// Dispositivo/Application/Pages/Schedulle
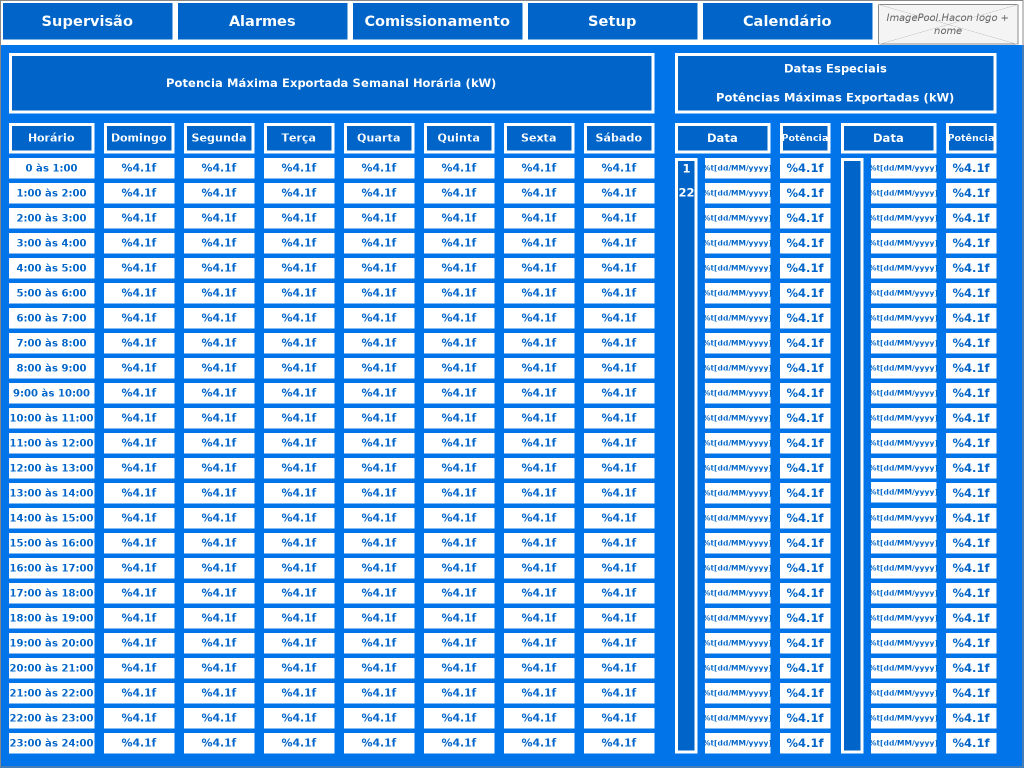
VISUALIZATION Schedulle  // 1024x768
    Frame (0,0 1024x768)
        shows Template()
    Rectangle (675,53 321x60), "Datas Especiais Potências Máximas Exportadas (kW)"
        OnMouseClick:  Assign=Setup, Type=Assignment
    Rectangle (104,123 70x30), "Domingo"
        OnMouseClick:  Assign=Setup, Type=Assignment
    Rectangle (104,158 70x20), "%4.1f", text variable: PerVar.WeekSchedule_kW[1,1]
        OnMouseEnter: write the text variable via Default, min 0, max 5000
    Rectangle (104,183 70x20), "%4.1f", text variable: PerVar.WeekSchedule_kW[1,2]
        OnMouseEnter: write the text variable via Default, min 0, max 5000
    Rectangle (104,208 70x20), "%4.1f", text variable: PerVar.WeekSchedule_kW[1,3]
        OnMouseEnter: write the text variable via Default, min 0, max 5000
    Rectangle (104,233 70x20), "%4.1f", text variable: PerVar.WeekSchedule_kW[1,4]
        OnMouseEnter: write the text variable via Default, min 0, max 5000
    Rectangle (104,258 70x20), "%4.1f", text variable: PerVar.WeekSchedule_kW[1,5]
        OnMouseEnter: write the text variable via Default, min 0, max 5000
    Rectangle (104,283 70x20), "%4.1f", text variable: PerVar.WeekSchedule_kW[1,6]
        OnMouseEnter: write the text variable via Default, min 0, max 5000
    Rectangle (104,308 70x20), "%4.1f", text variable: PerVar.WeekSchedule_kW[1,7]
        OnMouseEnter: write the text variable via Default, min 0, max 5000
    Rectangle (104,333 70x20), "%4.1f", text variable: PerVar.WeekSchedule_kW[1,8]
        OnMouseEnter: write the text variable via Default, min 0, max 5000
    Rectangle (104,358 70x20), "%4.1f", text variable: PerVar.WeekSchedule_kW[1,9]
        OnMouseEnter: write the text variable via Default, min 0, max 5000
    Rectangle (104,383 70x20), "%4.1f", text variable: PerVar.WeekSchedule_kW[1,10]
        OnMouseEnter: write the text variable via Default, min 0, max 5000
    Rectangle (104,408 70x20), "%4.1f", text variable: PerVar.WeekSchedule_kW[1,11]
        OnMouseEnter: write the text variable via Default, min 0, max 5000
    Rectangle (104,433 70x20), "%4.1f", text variable: PerVar.WeekSchedule_kW[1,12]
        OnMouseEnter: write the text variable via Default, min 0, max 5000
    Rectangle (104,458 70x20), "%4.1f", text variable: PerVar.WeekSchedule_kW[1,13]
        OnMouseEnter: write the text variable via Default, min 0, max 5000
    Rectangle (104,483 70x20), "%4.1f", text variable: PerVar.WeekSchedule_kW[1,14]
        OnMouseEnter: write the text variable via Default, min 0, max 5000
    Rectangle (104,508 70x20), "%4.1f", text variable: PerVar.WeekSchedule_kW[1,15]
        OnMouseEnter: write the text variable via Default, min 0, max 5000
    Rectangle (104,533 70x20), "%4.1f", text variable: PerVar.WeekSchedule_kW[1,16]
        OnMouseEnter: write the text variable via Default, min 0, max 5000
    Rectangle (104,558 70x20), "%4.1f", text variable: PerVar.WeekSchedule_kW[1,17]
        OnMouseEnter: write the text variable via Default, min 0, max 5000
    Rectangle (104,583 70x20), "%4.1f", text variable: PerVar.WeekSchedule_kW[1,18]
        OnMouseEnter: write the text variable via Default, min 0, max 5000
    Rectangle (104,608 70x20), "%4.1f", text variable: PerVar.WeekSchedule_kW[1,19]
        OnMouseEnter: write the text variable via Default, min 0, max 5000
    Rectangle (104,633 70x20), "%4.1f", text variable: PerVar.WeekSchedule_kW[1,20]
        OnMouseEnter: write the text variable via Default, min 0, max 5000
    Rectangle (104,658 70x20), "%4.1f", text variable: PerVar.WeekSchedule_kW[1,21]
        OnMouseEnter: write the text variable via Default, min 0, max 5000
    Rectangle (104,683 70x20), "%4.1f", text variable: PerVar.WeekSchedule_kW[1,22]
        OnMouseEnter: write the text variable via Default, min 0, max 5000
    Rectangle (104,708 70x20), "%4.1f", text variable: PerVar.WeekSchedule_kW[1,23]
        OnMouseEnter: write the text variable via Default, min 0, max 5000
    Rectangle (104,733 70x20), "%4.1f", text variable: PerVar.WeekSchedule_kW[1,24]
        OnMouseEnter: write the text variable via Default, min 0, max 5000
    Rectangle (705,158 65x20), "%t[dd/MM/yyyy]", tooltip "XX/XX/XXXX", text variable: PerVar.DatasEspeciais[1]
        OnMouseClick: write the text variable via Edit
    Rectangle (675,123 95x30), "Data"
        OnMouseClick:  Assign=Setup, Type=Assignment
    Rectangle (705,183 65x20), "%t[dd/MM/yyyy]", tooltip "XX/XX/XXXX", text variable: PerVar.DatasEspeciais[2]
        OnMouseClick: write the text variable via Edit
    Rectangle (705,208 65x20), "%t[dd/MM/yyyy]", tooltip "XX/XX/XXXX", text variable: PerVar.DatasEspeciais[3]
        OnMouseClick: write the text variable via Edit
    Rectangle (705,233 65x20), "%t[dd/MM/yyyy]", tooltip "XX/XX/XXXX", text variable: PerVar.DatasEspeciais[4]
        OnMouseClick: write the text variable via Edit
    Rectangle (705,258 65x20), "%t[dd/MM/yyyy]", tooltip "XX/XX/XXXX", text variable: PerVar.DatasEspeciais[5]
        OnMouseClick: write the text variable via Edit
    Rectangle (705,283 65x20), "%t[dd/MM/yyyy]", tooltip "XX/XX/XXXX", text variable: PerVar.DatasEspeciais[6]
        OnMouseClick: write the text variable via Edit
    Rectangle (705,308 65x20), "%t[dd/MM/yyyy]", tooltip "XX/XX/XXXX", text variable: PerVar.DatasEspeciais[7]
        OnMouseClick: write the text variable via Edit
    Rectangle (705,333 65x20), "%t[dd/MM/yyyy]", tooltip "XX/XX/XXXX", text variable: PerVar.DatasEspeciais[8]
        OnMouseClick: write the text variable via Edit
    Rectangle (705,358 65x20), "%t[dd/MM/yyyy]", tooltip "XX/XX/XXXX", text variable: PerVar.DatasEspeciais[9]
        OnMouseClick: write the text variable via Edit
    Rectangle (705,383 65x20), "%t[dd/MM/yyyy]", tooltip "XX/XX/XXXX", text variable: PerVar.DatasEspeciais[10]
        OnMouseClick: write the text variable via Edit
    Rectangle (705,408 65x20), "%t[dd/MM/yyyy]", tooltip "XX/XX/XXXX", text variable: PerVar.DatasEspeciais[11]
        OnMouseClick: write the text variable via Edit
    Rectangle (705,433 65x20), "%t[dd/MM/yyyy]", tooltip "XX/XX/XXXX", text variable: PerVar.DatasEspeciais[12]
        OnMouseClick: write the text variable via Edit
    Rectangle (705,458 65x20), "%t[dd/MM/yyyy]", tooltip "XX/XX/XXXX", text variable: PerVar.DatasEspeciais[13]
        OnMouseClick: write the text variable via Edit
    Rectangle (705,483 65x20), "%t[dd/MM/yyyy]", tooltip "XX/XX/XXXX", text variable: PerVar.DatasEspeciais[14]
        OnMouseClick: write the text variable via Edit
    Rectangle (705,508 65x20), "%t[dd/MM/yyyy]", tooltip "XX/XX/XXXX", text variable: PerVar.DatasEspeciais[15]
        OnMouseClick: write the text variable via Edit
    Rectangle (841,123 95x30), "Data"
        OnMouseClick:  Assign=Setup, Type=Assignment
    Rectangle (871,158 65x20), "%t[dd/MM/yyyy]", tooltip "XX/XX/XXXX", text variable: PerVar.DatasEspeciais[25]
        OnMouseClick: write the text variable via Edit
    Rectangle (871,183 65x20), "%t[dd/MM/yyyy]", tooltip "XX/XX/XXXX", text variable: PerVar.DatasEspeciais[26]
        OnMouseClick: write the text variable via Edit
    Rectangle (871,208 65x20), "%t[dd/MM/yyyy]", tooltip "XX/XX/XXXX", text variable: PerVar.DatasEspeciais[27]
        OnMouseClick: write the text variable via Edit
    Rectangle (871,233 65x20), "%t[dd/MM/yyyy]", tooltip "XX/XX/XXXX", text variable: PerVar.DatasEspeciais[28]
        OnMouseClick: write the text variable via Edit
    Rectangle (871,258 65x20), "%t[dd/MM/yyyy]", tooltip "XX/XX/XXXX", text variable: PerVar.DatasEspeciais[29]
        OnMouseClick: write the text variable via Edit
    Rectangle (871,283 65x20), "%t[dd/MM/yyyy]", tooltip "XX/XX/XXXX", text variable: PerVar.DatasEspeciais[30]
        OnMouseClick: write the text variable via Edit
    Rectangle (871,308 65x20), "%t[dd/MM/yyyy]", tooltip "XX/XX/XXXX", text variable: PerVar.DatasEspeciais[31]
        OnMouseClick: write the text variable via Edit
    Rectangle (871,333 65x20), "%t[dd/MM/yyyy]", tooltip "XX/XX/XXXX", text variable: PerVar.DatasEspeciais[32]
        OnMouseClick: write the text variable via Edit
    Rectangle (871,358 65x20), "%t[dd/MM/yyyy]", tooltip "XX/XX/XXXX", text variable: PerVar.DatasEspeciais[33]
        OnMouseClick: write the text variable via Edit
    Rectangle (871,383 65x20), "%t[dd/MM/yyyy]", tooltip "XX/XX/XXXX", text variable: PerVar.DatasEspeciais[34]
        OnMouseClick: write the text variable via Edit
    Rectangle (871,408 65x20), "%t[dd/MM/yyyy]", tooltip "XX/XX/XXXX", text variable: PerVar.DatasEspeciais[35]
        OnMouseClick: write the text variable via Edit
    Rectangle (871,433 65x20), "%t[dd/MM/yyyy]", tooltip "XX/XX/XXXX", text variable: PerVar.DatasEspeciais[36]
        OnMouseClick: write the text variable via Edit
    Rectangle (871,458 65x20), "%t[dd/MM/yyyy]", tooltip "XX/XX/XXXX", text variable: PerVar.DatasEspeciais[37]
        OnMouseClick: write the text variable via Edit
    Rectangle (871,482 65x20), "%t[dd/MM/yyyy]", tooltip "XX/XX/XXXX", text variable: PerVar.DatasEspeciais[38]
        OnMouseClick: write the text variable via Edit
    Rectangle (871,508 65x20), "%t[dd/MM/yyyy]", tooltip "XX/XX/XXXX", text variable: PerVar.DatasEspeciais[39]
        OnMouseClick: write the text variable via Edit
    Rectangle (780,123 50x30), "Potência"
        OnMouseClick:  Assign=Setup, Type=Assignment
    Rectangle (780,158 50x20), "%4.1f", text variable: PerVar.SpecialDaySchedule[1]
        OnMouseEnter: write the text variable via Default, min 0, max 5000
    Rectangle (780,183 50x20), "%4.1f", text variable: PerVar.SpecialDaySchedule[2]
        OnMouseEnter: write the text variable via Default, min 0, max 5000
    Rectangle (780,208 50x20), "%4.1f", text variable: PerVar.SpecialDaySchedule[3]
        OnMouseEnter: write the text variable via Default, min 0, max 5000
    Rectangle (780,233 50x20), "%4.1f", text variable: PerVar.SpecialDaySchedule[4]
        OnMouseEnter: write the text variable via Default, min 0, max 5000
    Rectangle (780,258 50x20), "%4.1f", text variable: PerVar.SpecialDaySchedule[5]
        OnMouseEnter: write the text variable via Default, min 0, max 5000
    Rectangle (780,283 50x20), "%4.1f", text variable: PerVar.SpecialDaySchedule[6]
        OnMouseEnter: write the text variable via Default, min 0, max 5000
    Rectangle (780,308 50x20), "%4.1f", text variable: PerVar.SpecialDaySchedule[7]
        OnMouseEnter: write the text variable via Default, min 0, max 5000
    Rectangle (780,333 50x20), "%4.1f", text variable: PerVar.SpecialDaySchedule[8]
        OnMouseEnter: write the text variable via Default, min 0, max 5000
    Rectangle (780,358 50x20), "%4.1f", text variable: PerVar.SpecialDaySchedule[9]
        OnMouseEnter: write the text variable via Default, min 0, max 5000
    Rectangle (780,383 50x20), "%4.1f", text variable: PerVar.SpecialDaySchedule[10]
        OnMouseEnter: write the text variable via Default, min 0, max 5000
    Rectangle (780,408 50x20), "%4.1f", text variable: PerVar.SpecialDaySchedule[11]
        OnMouseEnter: write the text variable via Default, min 0, max 5000
    Rectangle (780,433 50x20), "%4.1f", text variable: PerVar.SpecialDaySchedule[12]
        OnMouseEnter: write the text variable via Default, min 0, max 5000
    Rectangle (780,458 50x20), "%4.1f", text variable: PerVar.SpecialDaySchedule[13]
        OnMouseEnter: write the text variable via Default, min 0, max 5000
    Rectangle (780,483 50x20), "%4.1f", text variable: PerVar.SpecialDaySchedule[14]
        OnMouseEnter: write the text variable via Default, min 0, max 5000
    Rectangle (780,508 50x20), "%4.1f", text variable: PerVar.SpecialDaySchedule[15]
        OnMouseEnter: write the text variable via Default, min 0, max 5000
    Rectangle (780,533 50x20), "%4.1f", text variable: PerVar.SpecialDaySchedule[16]
        OnMouseEnter: write the text variable via Default, min 0, max 5000
    Rectangle (780,558 50x20), "%4.1f", text variable: PerVar.SpecialDaySchedule[17]
        OnMouseEnter: write the text variable via Default, min 0, max 5000
    Rectangle (780,583 50x20), "%4.1f", text variable: PerVar.SpecialDaySchedule[18]
        OnMouseEnter: write the text variable via Default, min 0, max 5000
    Rectangle (780,608 50x20), "%4.1f", text variable: PerVar.SpecialDaySchedule[19]
        OnMouseEnter: write the text variable via Default, min 0, max 5000
    Rectangle (780,633 50x20), "%4.1f", text variable: PerVar.SpecialDaySchedule[20]
        OnMouseEnter: write the text variable via Default, min 0, max 5000
    Rectangle (780,658 50x20), "%4.1f", text variable: PerVar.SpecialDaySchedule[21]
        OnMouseEnter: write the text variable via Default, min 0, max 5000
    Rectangle (780,683 50x20), "%4.1f", text variable: PerVar.SpecialDaySchedule[22]
        OnMouseEnter: write the text variable via Default, min 0, max 5000
    Rectangle (780,708 50x20), "%4.1f", text variable: PerVar.SpecialDaySchedule[23]
        OnMouseEnter: write the text variable via Default, min 0, max 5000
    Rectangle (780,733 50x20), "%4.1f", text variable: PerVar.SpecialDaySchedule[24]
        OnMouseEnter: write the text variable via Default, min 0, max 5000
    Rectangle (946,158 50x20), "%4.1f", text variable: PerVar.SpecialDaySchedule[25]
        OnMouseEnter: write the text variable via Default, min 0, max 5000
    Rectangle (946,183 50x20), "%4.1f", text variable: PerVar.SpecialDaySchedule[26]
        OnMouseEnter: write the text variable via Default, min 0, max 5000
    Rectangle (946,208 50x20), "%4.1f", text variable: PerVar.SpecialDaySchedule[27]
        OnMouseEnter: write the text variable via Default, min 0, max 5000
    Rectangle (946,233 50x20), "%4.1f", text variable: PerVar.SpecialDaySchedule[28]
        OnMouseEnter: write the text variable via Default, min 0, max 5000
    Rectangle (946,258 50x20), "%4.1f", text variable: PerVar.SpecialDaySchedule[29]
        OnMouseEnter: write the text variable via Default, min 0, max 5000
    Rectangle (946,283 50x20), "%4.1f", text variable: PerVar.SpecialDaySchedule[30]
        OnMouseEnter: write the text variable via Default, min 0, max 5000
    Rectangle (705,533 65x20), "%t[dd/MM/yyyy]", tooltip "XX/XX/XXXX", text variable: PerVar.DatasEspeciais[16]
        OnMouseClick: write the text variable via Edit
    Rectangle (705,558 65x20), "%t[dd/MM/yyyy]", tooltip "XX/XX/XXXX", text variable: PerVar.DatasEspeciais[17]
        OnMouseClick: write the text variable via Edit
    Rectangle (705,583 65x20), "%t[dd/MM/yyyy]", tooltip "XX/XX/XXXX", text variable: PerVar.DatasEspeciais[18]
        OnMouseClick: write the text variable via Edit
    Rectangle (705,608 65x20), "%t[dd/MM/yyyy]", tooltip "XX/XX/XXXX", text variable: PerVar.DatasEspeciais[19]
        OnMouseClick: write the text variable via Edit
    Rectangle (705,633 65x20), "%t[dd/MM/yyyy]", tooltip "XX/XX/XXXX", text variable: PerVar.DatasEspeciais[20]
        OnMouseClick: write the text variable via Edit
    Rectangle (705,658 65x20), "%t[dd/MM/yyyy]", tooltip "XX/XX/XXXX", text variable: PerVar.DatasEspeciais[21]
        OnMouseClick: write the text variable via Edit
    Rectangle (705,683 65x20), "%t[dd/MM/yyyy]", tooltip "XX/XX/XXXX", text variable: PerVar.DatasEspeciais[22]
        OnMouseClick: write the text variable via Edit
    Rectangle (705,708 65x20), "%t[dd/MM/yyyy]", tooltip "XX/XX/XXXX", text variable: PerVar.DatasEspeciais[23]
        OnMouseClick: write the text variable via Edit
    Rectangle (705,733 65x20), "%t[dd/MM/yyyy]", tooltip "XX/XX/XXXX", text variable: PerVar.DatasEspeciais[24]
        OnMouseClick: write the text variable via Edit
    Rectangle (871,533 65x20), "%t[dd/MM/yyyy]", tooltip "XX/XX/XXXX", text variable: PerVar.DatasEspeciais[40]
        OnMouseClick: write the text variable via Edit
    Rectangle (871,558 65x20), "%t[dd/MM/yyyy]", tooltip "XX/XX/XXXX", text variable: PerVar.DatasEspeciais[41]
        OnMouseClick: write the text variable via Edit
    Rectangle (871,583 65x20), "%t[dd/MM/yyyy]", tooltip "XX/XX/XXXX", text variable: PerVar.DatasEspeciais[42]
        OnMouseClick: write the text variable via Edit
    Rectangle (871,608 65x20), "%t[dd/MM/yyyy]", tooltip "XX/XX/XXXX", text variable: PerVar.DatasEspeciais[43]
        OnMouseClick: write the text variable via Edit
    Rectangle (871,633 65x20), "%t[dd/MM/yyyy]", tooltip "XX/XX/XXXX", text variable: PerVar.DatasEspeciais[44]
        OnMouseClick: write the text variable via Edit
    Rectangle (871,658 65x20), "%t[dd/MM/yyyy]", tooltip "XX/XX/XXXX", text variable: PerVar.DatasEspeciais[45]
        OnMouseClick: write the text variable via Edit
    Rectangle (871,683 65x20), "%t[dd/MM/yyyy]", tooltip "XX/XX/XXXX", text variable: PerVar.DatasEspeciais[46]
        OnMouseClick: write the text variable via Edit
    Rectangle (871,708 65x20), "%t[dd/MM/yyyy]", tooltip "XX/XX/XXXX", text variable: PerVar.DatasEspeciais[47]
        OnMouseClick: write the text variable via Edit
    Rectangle (871,733 65x20), "%t[dd/MM/yyyy]", tooltip "XX/XX/XXXX", text variable: PerVar.DatasEspeciais[48]
        OnMouseClick: write the text variable via Edit
    Rectangle (946,308 50x20), "%4.1f", text variable: PerVar.SpecialDaySchedule[31]
        OnMouseEnter: write the text variable via Default, min 0, max 5000
    Rectangle (946,333 50x20), "%4.1f", text variable: PerVar.SpecialDaySchedule[32]
        OnMouseEnter: write the text variable via Default, min 0, max 5000
    Rectangle (946,358 50x20), "%4.1f", text variable: PerVar.SpecialDaySchedule[33]
        OnMouseEnter: write the text variable via Default, min 0, max 5000
    Rectangle (946,383 50x20), "%4.1f", text variable: PerVar.SpecialDaySchedule[34]
        OnMouseEnter: write the text variable via Default, min 0, max 5000
    Rectangle (946,408 50x20), "%4.1f", text variable: PerVar.SpecialDaySchedule[35]
        OnMouseEnter: write the text variable via Default, min 0, max 5000
    Rectangle (946,433 50x20), "%4.1f", text variable: PerVar.SpecialDaySchedule[36]
        OnMouseEnter: write the text variable via Default, min 0, max 5000
    Rectangle (946,458 50x20), "%4.1f", text variable: PerVar.SpecialDaySchedule[37]
        OnMouseEnter: write the text variable via Default, min 0, max 5000
    Rectangle (946,483 50x20), "%4.1f", text variable: PerVar.SpecialDaySchedule[38]
        OnMouseEnter: write the text variable via Default, min 0, max 5000
    Rectangle (946,508 50x20), "%4.1f", text variable: PerVar.SpecialDaySchedule[39]
        OnMouseEnter: write the text variable via Default, min 0, max 5000
    Rectangle (946,533 50x20), "%4.1f", text variable: PerVar.SpecialDaySchedule[40]
        OnMouseEnter: write the text variable via Default, min 0, max 5000
    Rectangle (946,558 50x20), "%4.1f", text variable: PerVar.SpecialDaySchedule[41]
        OnMouseEnter: write the text variable via Default, min 0, max 5000
    Rectangle (946,583 50x20), "%4.1f", text variable: PerVar.SpecialDaySchedule[42]
        OnMouseEnter: write the text variable via Default, min 0, max 5000
    Rectangle (946,608 50x20), "%4.1f", text variable: PerVar.SpecialDaySchedule[43]
        OnMouseEnter: write the text variable via Default, min 0, max 5000
    Rectangle (946,633 50x20), "%4.1f", text variable: PerVar.SpecialDaySchedule[44]
        OnMouseEnter: write the text variable via Default, min 0, max 5000
    Rectangle (946,658 50x20), "%4.1f", text variable: PerVar.SpecialDaySchedule[45]
        OnMouseEnter: write the text variable via Default, min 0, max 5000
    Rectangle (946,683 50x20), "%4.1f", text variable: PerVar.SpecialDaySchedule[46]
        OnMouseEnter: write the text variable via Default, min 0, max 5000
    Rectangle (946,708 50x20), "%4.1f", text variable: PerVar.SpecialDaySchedule[47]
        OnMouseEnter: write the text variable via Default, min 0, max 5000
    Rectangle (946,733 50x20), "%4.1f", text variable: PerVar.SpecialDaySchedule[48]
        OnMouseEnter: write the text variable via Default, min 0, max 5000
    Rectangle (9,53 645x60), "Potencia Máxima Exportada Semanal Horária (kW)"
        OnMouseClick:  Assign=Setup, Type=Assignment
    Rectangle (184,123 70x30), "Segunda"
        OnMouseClick:  Assign=Setup, Type=Assignment
    Rectangle (264,123 70x30), "Terça"
        OnMouseClick:  Assign=Setup, Type=Assignment
    Rectangle (344,123 70x30), "Quarta"
        OnMouseClick:  Assign=Setup, Type=Assignment
    Rectangle (424,123 70x30), "Quinta"
        OnMouseClick:  Assign=Setup, Type=Assignment
    Rectangle (504,123 70x30), "Sexta"
        OnMouseClick:  Assign=Setup, Type=Assignment
    Rectangle (584,123 70x30), "Sábado"
        OnMouseClick:  Assign=Setup, Type=Assignment
    Rectangle (9,158 85x20), "0 às 1:00"
    Rectangle (9,123 85x30), "Horário"
        OnMouseClick:  Assign=Setup, Type=Assignment
    Rectangle (9,183 85x20), "1:00 às 2:00"
    Rectangle (9,208 85x20), "2:00 às 3:00"
    Rectangle (9,233 85x20), "3:00 às 4:00"
    Rectangle (9,258 85x20), "4:00 às 5:00"
    Rectangle (9,283 85x20), "5:00 às 6:00"
    Rectangle (9,308 85x20), "6:00 às 7:00"
    Rectangle (9,333 85x20), "7:00 às 8:00"
    Rectangle (9,358 85x20), "8:00 às 9:00"
    Rectangle (9,383 85x20), "9:00 às 10:00"
    Rectangle (9,408 85x20), "10:00 às 11:00"
    Rectangle (9,433 85x20), "11:00 às 12:00"
    Rectangle (9,458 85x20), "12:00 às 13:00"
    Rectangle (9,483 85x20), "13:00 às 14:00"
    Rectangle (9,508 85x20), "14:00 às 15:00"
    Rectangle (9,533 85x20), "15:00 às 16:00"
    Rectangle (9,558 85x20), "16:00 às 17:00"
    Rectangle (9,583 85x20), "17:00 às 18:00"
    Rectangle (9,608 85x20), "18:00 às 19:00"
    Rectangle (9,633 85x20), "19:00 às 20:00"
    Rectangle (9,658 85x20), "20:00 às 21:00"
    Rectangle (9,683 85x20), "21:00 às 22:00"
    Rectangle (9,708 85x20), "22:00 às 23:00"
    Rectangle (9,733 85x20), "23:00 às 24:00"
    Rectangle (184,158 70x20), "%4.1f", text variable: PerVar.WeekSchedule_kW[2,1]
        OnMouseEnter: write the text variable via Default, min 0, max 5000
    Rectangle (184,183 70x20), "%4.1f", text variable: PerVar.WeekSchedule_kW[2,2]
        OnMouseEnter: write the text variable via Default, min 0, max 5000
    Rectangle (184,208 70x20), "%4.1f", text variable: PerVar.WeekSchedule_kW[2,3]
        OnMouseEnter: write the text variable via Default, min 0, max 5000
    Rectangle (184,233 70x20), "%4.1f", text variable: PerVar.WeekSchedule_kW[2,4]
        OnMouseEnter: write the text variable via Default, min 0, max 5000
    Rectangle (184,258 70x20), "%4.1f", text variable: PerVar.WeekSchedule_kW[2,5]
        OnMouseEnter: write the text variable via Default, min 0, max 5000
    Rectangle (184,283 70x20), "%4.1f", text variable: PerVar.WeekSchedule_kW[2,6]
        OnMouseEnter: write the text variable via Default, min 0, max 5000
    Rectangle (184,308 70x20), "%4.1f", text variable: PerVar.WeekSchedule_kW[2,7]
        OnMouseEnter: write the text variable via Default, min 0, max 5000
    Rectangle (184,333 70x20), "%4.1f", text variable: PerVar.WeekSchedule_kW[2,8]
        OnMouseEnter: write the text variable via Default, min 0, max 5000
    Rectangle (184,358 70x20), "%4.1f", text variable: PerVar.WeekSchedule_kW[2,9]
        OnMouseEnter: write the text variable via Default, min 0, max 5000
    Rectangle (184,383 70x20), "%4.1f", text variable: PerVar.WeekSchedule_kW[2,10]
        OnMouseEnter: write the text variable via Default, min 0, max 5000
    Rectangle (184,408 70x20), "%4.1f", text variable: PerVar.WeekSchedule_kW[2,11]
        OnMouseEnter: write the text variable via Default, min 0, max 5000
    Rectangle (184,433 70x20), "%4.1f", text variable: PerVar.WeekSchedule_kW[2,12]
        OnMouseEnter: write the text variable via Default, min 0, max 5000
    Rectangle (184,458 70x20), "%4.1f", text variable: PerVar.WeekSchedule_kW[2,13]
        OnMouseEnter: write the text variable via Default, min 0, max 5000
    Rectangle (184,483 70x20), "%4.1f", text variable: PerVar.WeekSchedule_kW[2,14]
        OnMouseEnter: write the text variable via Default, min 0, max 5000
    Rectangle (184,508 70x20), "%4.1f", text variable: PerVar.WeekSchedule_kW[2,15]
        OnMouseEnter: write the text variable via Default, min 0, max 5000
    Rectangle (184,533 70x20), "%4.1f", text variable: PerVar.WeekSchedule_kW[2,16]
        OnMouseEnter: write the text variable via Default, min 0, max 5000
    Rectangle (184,558 70x20), "%4.1f", text variable: PerVar.WeekSchedule_kW[2,17]
        OnMouseEnter: write the text variable via Default, min 0, max 5000
    Rectangle (184,583 70x20), "%4.1f", text variable: PerVar.WeekSchedule_kW[2,18]
        OnMouseEnter: write the text variable via Default, min 0, max 5000
    Rectangle (184,608 70x20), "%4.1f", text variable: PerVar.WeekSchedule_kW[2,19]
        OnMouseEnter: write the text variable via Default, min 0, max 5000
    Rectangle (184,633 70x20), "%4.1f", text variable: PerVar.WeekSchedule_kW[2,20]
        OnMouseEnter: write the text variable via Default, min 0, max 5000
    Rectangle (184,658 70x20), "%4.1f", text variable: PerVar.WeekSchedule_kW[2,21]
        OnMouseEnter: write the text variable via Default, min 0, max 5000
    Rectangle (184,683 70x20), "%4.1f", text variable: PerVar.WeekSchedule_kW[2,22]
        OnMouseEnter: write the text variable via Default, min 0, max 5000
    Rectangle (184,708 70x20), "%4.1f", text variable: PerVar.WeekSchedule_kW[2,23]
        OnMouseEnter: write the text variable via Default, min 0, max 5000
    Rectangle (184,733 70x20), "%4.1f", text variable: PerVar.WeekSchedule_kW[2,24]
        OnMouseEnter: write the text variable via Default, min 0, max 5000
    Rectangle (344,158 70x20), "%4.1f", text variable: PerVar.WeekSchedule_kW[4,1]
        OnMouseEnter: write the text variable via Default, min 0, max 5000
    Rectangle (344,183 70x20), "%4.1f", text variable: PerVar.WeekSchedule_kW[4,2]
        OnMouseEnter: write the text variable via Default, min 0, max 5000
    Rectangle (344,208 70x20), "%4.1f", text variable: PerVar.WeekSchedule_kW[4,3]
        OnMouseEnter: write the text variable via Default, min 0, max 5000
    Rectangle (344,233 70x20), "%4.1f", text variable: PerVar.WeekSchedule_kW[4,4]
        OnMouseEnter: write the text variable via Default, min 0, max 5000
    Rectangle (344,258 70x20), "%4.1f", text variable: PerVar.WeekSchedule_kW[4,5]
        OnMouseEnter: write the text variable via Default, min 0, max 5000
    Rectangle (344,283 70x20), "%4.1f", text variable: PerVar.WeekSchedule_kW[4,6]
        OnMouseEnter: write the text variable via Default, min 0, max 5000
    Rectangle (344,308 70x20), "%4.1f", text variable: PerVar.WeekSchedule_kW[4,7]
        OnMouseEnter: write the text variable via Default, min 0, max 5000
    Rectangle (344,333 70x20), "%4.1f", text variable: PerVar.WeekSchedule_kW[4,8]
        OnMouseEnter: write the text variable via Default, min 0, max 5000
    Rectangle (344,358 70x20), "%4.1f", text variable: PerVar.WeekSchedule_kW[4,9]
        OnMouseEnter: write the text variable via Default, min 0, max 5000
    Rectangle (344,383 70x20), "%4.1f", text variable: PerVar.WeekSchedule_kW[4,10]
        OnMouseEnter: write the text variable via Default, min 0, max 5000
    Rectangle (344,408 70x20), "%4.1f", text variable: PerVar.WeekSchedule_kW[4,11]
        OnMouseEnter: write the text variable via Default, min 0, max 5000
    Rectangle (344,433 70x20), "%4.1f", text variable: PerVar.WeekSchedule_kW[4,12]
        OnMouseEnter: write the text variable via Default, min 0, max 5000
    Rectangle (344,458 70x20), "%4.1f", text variable: PerVar.WeekSchedule_kW[4,13]
        OnMouseEnter: write the text variable via Default, min 0, max 5000
    Rectangle (344,483 70x20), "%4.1f", text variable: PerVar.WeekSchedule_kW[4,14]
        OnMouseEnter: write the text variable via Default, min 0, max 5000
    Rectangle (344,508 70x20), "%4.1f", text variable: PerVar.WeekSchedule_kW[4,15]
        OnMouseEnter: write the text variable via Default, min 0, max 5000
    Rectangle (344,533 70x20), "%4.1f", text variable: PerVar.WeekSchedule_kW[4,16]
        OnMouseEnter: write the text variable via Default, min 0, max 5000
    Rectangle (344,558 70x20), "%4.1f", text variable: PerVar.WeekSchedule_kW[4,17]
        OnMouseEnter: write the text variable via Default, min 0, max 5000
    Rectangle (344,583 70x20), "%4.1f", text variable: PerVar.WeekSchedule_kW[4,18]
        OnMouseEnter: write the text variable via Default, min 0, max 5000
    Rectangle (344,608 70x20), "%4.1f", text variable: PerVar.WeekSchedule_kW[4,19]
        OnMouseEnter: write the text variable via Default, min 0, max 5000
    Rectangle (344,633 70x20), "%4.1f", text variable: PerVar.WeekSchedule_kW[4,20]
        OnMouseEnter: write the text variable via Default, min 0, max 5000
    Rectangle (344,658 70x20), "%4.1f", text variable: PerVar.WeekSchedule_kW[4,21]
        OnMouseEnter: write the text variable via Default, min 0, max 5000
    Rectangle (344,683 70x20), "%4.1f", text variable: PerVar.WeekSchedule_kW[4,22]
        OnMouseEnter: write the text variable via Default, min 0, max 5000
    Rectangle (344,708 70x20), "%4.1f", text variable: PerVar.WeekSchedule_kW[4,23]
        OnMouseEnter: write the text variable via Default, min 0, max 5000
    Rectangle (344,733 70x20), "%4.1f", text variable: PerVar.WeekSchedule_kW[4,24]
        OnMouseEnter: write the text variable via Default, min 0, max 5000
    Rectangle (264,158 70x20), "%4.1f", text variable: PerVar.WeekSchedule_kW[3,1]
        OnMouseEnter: write the text variable via Default, min 0, max 5000
    Rectangle (264,183 70x20), "%4.1f", text variable: PerVar.WeekSchedule_kW[3,2]
        OnMouseEnter: write the text variable via Default, min 0, max 5000
    Rectangle (264,208 70x20), "%4.1f", text variable: PerVar.WeekSchedule_kW[3,3]
        OnMouseEnter: write the text variable via Default, min 0, max 5000
    Rectangle (264,233 70x20), "%4.1f", text variable: PerVar.WeekSchedule_kW[3,4]
        OnMouseEnter: write the text variable via Default, min 0, max 5000
    Rectangle (264,258 70x20), "%4.1f", text variable: PerVar.WeekSchedule_kW[3,5]
        OnMouseEnter: write the text variable via Default, min 0, max 5000
    Rectangle (264,283 70x20), "%4.1f", text variable: PerVar.WeekSchedule_kW[3,6]
        OnMouseEnter: write the text variable via Default, min 0, max 5000
    Rectangle (264,308 70x20), "%4.1f", text variable: PerVar.WeekSchedule_kW[3,7]
        OnMouseEnter: write the text variable via Default, min 0, max 5000
    Rectangle (264,333 70x20), "%4.1f", text variable: PerVar.WeekSchedule_kW[3,8]
        OnMouseEnter: write the text variable via Default, min 0, max 5000
    Rectangle (264,358 70x20), "%4.1f", text variable: PerVar.WeekSchedule_kW[3,9]
        OnMouseEnter: write the text variable via Default, min 0, max 5000
    Rectangle (264,383 70x20), "%4.1f", text variable: PerVar.WeekSchedule_kW[3,10]
        OnMouseEnter: write the text variable via Default, min 0, max 5000
    Rectangle (264,408 70x20), "%4.1f", text variable: PerVar.WeekSchedule_kW[3,11]
        OnMouseEnter: write the text variable via Default, min 0, max 5000
    Rectangle (264,433 70x20), "%4.1f", text variable: PerVar.WeekSchedule_kW[3,12]
        OnMouseEnter: write the text variable via Default, min 0, max 5000
    Rectangle (264,458 70x20), "%4.1f", text variable: PerVar.WeekSchedule_kW[3,13]
        OnMouseEnter: write the text variable via Default, min 0, max 5000
    Rectangle (264,483 70x20), "%4.1f", text variable: PerVar.WeekSchedule_kW[3,14]
        OnMouseEnter: write the text variable via Default, min 0, max 5000
    Rectangle (264,508 70x20), "%4.1f", text variable: PerVar.WeekSchedule_kW[3,15]
        OnMouseEnter: write the text variable via Default, min 0, max 5000
    Rectangle (264,533 70x20), "%4.1f", text variable: PerVar.WeekSchedule_kW[3,16]
        OnMouseEnter: write the text variable via Default, min 0, max 5000
    Rectangle (264,558 70x20), "%4.1f", text variable: PerVar.WeekSchedule_kW[3,17]
        OnMouseEnter: write the text variable via Default, min 0, max 5000
    Rectangle (264,583 70x20), "%4.1f", text variable: PerVar.WeekSchedule_kW[3,18]
        OnMouseEnter: write the text variable via Default, min 0, max 5000
    Rectangle (264,608 70x20), "%4.1f", text variable: PerVar.WeekSchedule_kW[3,19]
        OnMouseEnter: write the text variable via Default, min 0, max 5000
    Rectangle (264,633 70x20), "%4.1f", text variable: PerVar.WeekSchedule_kW[3,20]
        OnMouseEnter: write the text variable via Default, min 0, max 5000
    Rectangle (264,658 70x20), "%4.1f", text variable: PerVar.WeekSchedule_kW[3,21]
        OnMouseEnter: write the text variable via Default, min 0, max 5000
    Rectangle (264,683 70x20), "%4.1f", text variable: PerVar.WeekSchedule_kW[3,22]
        OnMouseEnter: write the text variable via Default, min 0, max 5000
    Rectangle (264,708 70x20), "%4.1f", text variable: PerVar.WeekSchedule_kW[3,23]
        OnMouseEnter: write the text variable via Default, min 0, max 5000
    Rectangle (264,733 70x20), "%4.1f", text variable: PerVar.WeekSchedule_kW[3,24]
        OnMouseEnter: write the text variable via Default, min 0, max 5000
    Rectangle (424,158 70x20), "%4.1f", text variable: PerVar.WeekSchedule_kW[5,1]
        OnMouseEnter: write the text variable via Default, min 0, max 5000
    Rectangle (424,183 70x20), "%4.1f", text variable: PerVar.WeekSchedule_kW[5,2]
        OnMouseEnter: write the text variable via Default, min 0, max 5000
    Rectangle (424,208 70x20), "%4.1f", text variable: PerVar.WeekSchedule_kW[5,3]
        OnMouseEnter: write the text variable via Default, min 0, max 5000
    Rectangle (424,233 70x20), "%4.1f", text variable: PerVar.WeekSchedule_kW[5,4]
        OnMouseEnter: write the text variable via Default, min 0, max 5000
    Rectangle (424,258 70x20), "%4.1f", text variable: PerVar.WeekSchedule_kW[5,5]
        OnMouseEnter: write the text variable via Default, min 0, max 5000
    Rectangle (424,283 70x20), "%4.1f", text variable: PerVar.WeekSchedule_kW[5,6]
        OnMouseEnter: write the text variable via Default, min 0, max 5000
    Rectangle (424,308 70x20), "%4.1f", text variable: PerVar.WeekSchedule_kW[5,7]
        OnMouseEnter: write the text variable via Default, min 0, max 5000
    Rectangle (424,333 70x20), "%4.1f", text variable: PerVar.WeekSchedule_kW[5,8]
        OnMouseEnter: write the text variable via Default, min 0, max 5000
    Rectangle (424,358 70x20), "%4.1f", text variable: PerVar.WeekSchedule_kW[5,9]
        OnMouseEnter: write the text variable via Default, min 0, max 5000
    Rectangle (424,383 70x20), "%4.1f", text variable: PerVar.WeekSchedule_kW[5,10]
        OnMouseEnter: write the text variable via Default, min 0, max 5000
    Rectangle (424,408 70x20), "%4.1f", text variable: PerVar.WeekSchedule_kW[5,11]
        OnMouseEnter: write the text variable via Default, min 0, max 5000
    Rectangle (424,433 70x20), "%4.1f", text variable: PerVar.WeekSchedule_kW[5,12]
        OnMouseEnter: write the text variable via Default, min 0, max 5000
    Rectangle (424,458 70x20), "%4.1f", text variable: PerVar.WeekSchedule_kW[5,13]
        OnMouseEnter: write the text variable via Default, min 0, max 5000
    Rectangle (424,483 70x20), "%4.1f", text variable: PerVar.WeekSchedule_kW[5,14]
        OnMouseEnter: write the text variable via Default, min 0, max 5000
    Rectangle (424,508 70x20), "%4.1f", text variable: PerVar.WeekSchedule_kW[5,15]
        OnMouseEnter: write the text variable via Default, min 0, max 5000
    Rectangle (424,533 70x20), "%4.1f", text variable: PerVar.WeekSchedule_kW[5,16]
        OnMouseEnter: write the text variable via Default, min 0, max 5000
    Rectangle (424,558 70x20), "%4.1f", text variable: PerVar.WeekSchedule_kW[5,17]
        OnMouseEnter: write the text variable via Default, min 0, max 5000
    Rectangle (424,583 70x20), "%4.1f", text variable: PerVar.WeekSchedule_kW[5,18]
        OnMouseEnter: write the text variable via Default, min 0, max 5000
    Rectangle (424,608 70x20), "%4.1f", text variable: PerVar.WeekSchedule_kW[5,19]
        OnMouseEnter: write the text variable via Default, min 0, max 5000
    Rectangle (424,633 70x20), "%4.1f", text variable: PerVar.WeekSchedule_kW[5,20]
        OnMouseEnter: write the text variable via Default, min 0, max 5000
    Rectangle (424,658 70x20), "%4.1f", text variable: PerVar.WeekSchedule_kW[5,21]
        OnMouseEnter: write the text variable via Default, min 0, max 5000
    Rectangle (424,683 70x20), "%4.1f", text variable: PerVar.WeekSchedule_kW[5,22]
        OnMouseEnter: write the text variable via Default, min 0, max 5000
    Rectangle (424,708 70x20), "%4.1f", text variable: PerVar.WeekSchedule_kW[5,23]
        OnMouseEnter: write the text variable via Default, min 0, max 5000
    Rectangle (424,733 70x20), "%4.1f", text variable: PerVar.WeekSchedule_kW[5,24]
        OnMouseEnter: write the text variable via Default, min 0, max 5000
    Rectangle (504,158 70x20), "%4.1f", text variable: PerVar.WeekSchedule_kW[6,1]
        OnMouseEnter: write the text variable via Default, min 0, max 5000
    Rectangle (504,183 70x20), "%4.1f", text variable: PerVar.WeekSchedule_kW[6,2]
        OnMouseEnter: write the text variable via Default, min 0, max 5000
    Rectangle (504,208 70x20), "%4.1f", text variable: PerVar.WeekSchedule_kW[6,3]
        OnMouseEnter: write the text variable via Default, min 0, max 5000
    Rectangle (504,233 70x20), "%4.1f", text variable: PerVar.WeekSchedule_kW[6,4]
        OnMouseEnter: write the text variable via Default, min 0, max 5000
    Rectangle (504,258 70x20), "%4.1f", text variable: PerVar.WeekSchedule_kW[6,5]
        OnMouseEnter: write the text variable via Default, min 0, max 5000
    Rectangle (504,283 70x20), "%4.1f", text variable: PerVar.WeekSchedule_kW[6,6]
        OnMouseEnter: write the text variable via Default, min 0, max 5000
    Rectangle (504,308 70x20), "%4.1f", text variable: PerVar.WeekSchedule_kW[6,7]
        OnMouseEnter: write the text variable via Default, min 0, max 5000
    Rectangle (504,333 70x20), "%4.1f", text variable: PerVar.WeekSchedule_kW[6,8]
        OnMouseEnter: write the text variable via Default, min 0, max 5000
    Rectangle (504,358 70x20), "%4.1f", text variable: PerVar.WeekSchedule_kW[6,9]
        OnMouseEnter: write the text variable via Default, min 0, max 5000
    Rectangle (504,383 70x20), "%4.1f", text variable: PerVar.WeekSchedule_kW[6,10]
        OnMouseEnter: write the text variable via Default, min 0, max 5000
    Rectangle (504,408 70x20), "%4.1f", text variable: PerVar.WeekSchedule_kW[6,11]
        OnMouseEnter: write the text variable via Default, min 0, max 5000
    Rectangle (504,433 70x20), "%4.1f", text variable: PerVar.WeekSchedule_kW[6,12]
        OnMouseEnter: write the text variable via Default, min 0, max 5000
    Rectangle (504,458 70x20), "%4.1f", text variable: PerVar.WeekSchedule_kW[6,13]
        OnMouseEnter: write the text variable via Default, min 0, max 5000
    Rectangle (504,483 70x20), "%4.1f", text variable: PerVar.WeekSchedule_kW[6,14]
        OnMouseEnter: write the text variable via Default, min 0, max 5000
    Rectangle (504,508 70x20), "%4.1f", text variable: PerVar.WeekSchedule_kW[6,15]
        OnMouseEnter: write the text variable via Default, min 0, max 5000
    Rectangle (504,533 70x20), "%4.1f", text variable: PerVar.WeekSchedule_kW[6,16]
        OnMouseEnter: write the text variable via Default, min 0, max 5000
    Rectangle (504,558 70x20), "%4.1f", text variable: PerVar.WeekSchedule_kW[6,17]
        OnMouseEnter: write the text variable via Default, min 0, max 5000
    Rectangle (504,583 70x20), "%4.1f", text variable: PerVar.WeekSchedule_kW[6,18]
        OnMouseEnter: write the text variable via Default, min 0, max 5000
    Rectangle (504,608 70x20), "%4.1f", text variable: PerVar.WeekSchedule_kW[6,19]
        OnMouseEnter: write the text variable via Default, min 0, max 5000
    Rectangle (504,633 70x20), "%4.1f", text variable: PerVar.WeekSchedule_kW[6,20]
        OnMouseEnter: write the text variable via Default, min 0, max 5000
    Rectangle (504,658 70x20), "%4.1f", text variable: PerVar.WeekSchedule_kW[6,21]
        OnMouseEnter: write the text variable via Default, min 0, max 5000
    Rectangle (504,683 70x20), "%4.1f", text variable: PerVar.WeekSchedule_kW[6,22]
        OnMouseEnter: write the text variable via Default, min 0, max 5000
    Rectangle (504,708 70x20), "%4.1f", text variable: PerVar.WeekSchedule_kW[6,23]
        OnMouseEnter: write the text variable via Default, min 0, max 5000
    Rectangle (504,733 70x20), "%4.1f", text variable: PerVar.WeekSchedule_kW[6,24]
        OnMouseEnter: write the text variable via Default, min 0, max 5000
    Rectangle (584,158 70x20), "%4.1f", text variable: PerVar.WeekSchedule_kW[7,1]
        OnMouseEnter: write the text variable via Default, min 0, max 5000
    Rectangle (584,183 70x20), "%4.1f", text variable: PerVar.WeekSchedule_kW[7,2]
        OnMouseEnter: write the text variable via Default, min 0, max 5000
    Rectangle (584,208 70x20), "%4.1f", text variable: PerVar.WeekSchedule_kW[7,3]
        OnMouseEnter: write the text variable via Default, min 0, max 5000
    Rectangle (584,233 70x20), "%4.1f", text variable: PerVar.WeekSchedule_kW[7,4]
        OnMouseEnter: write the text variable via Default, min 0, max 5000
    Rectangle (584,258 70x20), "%4.1f", text variable: PerVar.WeekSchedule_kW[7,5]
        OnMouseEnter: write the text variable via Default, min 0, max 5000
    Rectangle (584,283 70x20), "%4.1f", text variable: PerVar.WeekSchedule_kW[7,6]
        OnMouseEnter: write the text variable via Default, min 0, max 5000
    Rectangle (584,308 70x20), "%4.1f", text variable: PerVar.WeekSchedule_kW[7,7]
        OnMouseEnter: write the text variable via Default, min 0, max 5000
    Rectangle (584,333 70x20), "%4.1f", text variable: PerVar.WeekSchedule_kW[7,8]
        OnMouseEnter: write the text variable via Default, min 0, max 5000
    Rectangle (584,358 70x20), "%4.1f", text variable: PerVar.WeekSchedule_kW[7,9]
        OnMouseEnter: write the text variable via Default, min 0, max 5000
    Rectangle (584,383 70x20), "%4.1f", text variable: PerVar.WeekSchedule_kW[7,10]
        OnMouseEnter: write the text variable via Default, min 0, max 5000
    Rectangle (584,408 70x20), "%4.1f", text variable: PerVar.WeekSchedule_kW[7,11]
        OnMouseEnter: write the text variable via Default, min 0, max 5000
    Rectangle (584,433 70x20), "%4.1f", text variable: PerVar.WeekSchedule_kW[7,12]
        OnMouseEnter: write the text variable via Default, min 0, max 5000
    Rectangle (584,458 70x20), "%4.1f", text variable: PerVar.WeekSchedule_kW[7,13]
        OnMouseEnter: write the text variable via Default, min 0, max 5000
    Rectangle (584,483 70x20), "%4.1f", text variable: PerVar.WeekSchedule_kW[7,14]
        OnMouseEnter: write the text variable via Default, min 0, max 5000
    Rectangle (584,508 70x20), "%4.1f", text variable: PerVar.WeekSchedule_kW[7,15]
        OnMouseEnter: write the text variable via Default, min 0, max 5000
    Rectangle (584,533 70x20), "%4.1f", text variable: PerVar.WeekSchedule_kW[7,16]
        OnMouseEnter: write the text variable via Default, min 0, max 5000
    Rectangle (584,558 70x20), "%4.1f", text variable: PerVar.WeekSchedule_kW[7,17]
        OnMouseEnter: write the text variable via Default, min 0, max 5000
    Rectangle (584,583 70x20), "%4.1f", text variable: PerVar.WeekSchedule_kW[7,18]
        OnMouseEnter: write the text variable via Default, min 0, max 5000
    Rectangle (584,608 70x20), "%4.1f", text variable: PerVar.WeekSchedule_kW[7,19]
        OnMouseEnter: write the text variable via Default, min 0, max 5000
    Rectangle (584,633 70x20), "%4.1f", text variable: PerVar.WeekSchedule_kW[7,20]
        OnMouseEnter: write the text variable via Default, min 0, max 5000
    Rectangle (584,658 70x20), "%4.1f", text variable: PerVar.WeekSchedule_kW[7,21]
        OnMouseEnter: write the text variable via Default, min 0, max 5000
    Rectangle (584,683 70x20), "%4.1f", text variable: PerVar.WeekSchedule_kW[7,22]
        OnMouseEnter: write the text variable via Default, min 0, max 5000
    Rectangle (584,708 70x20), "%4.1f", text variable: PerVar.WeekSchedule_kW[7,23]
        OnMouseEnter: write the text variable via Default, min 0, max 5000
    Rectangle (584,733 70x20), "%4.1f", text variable: PerVar.WeekSchedule_kW[7,24]
        OnMouseEnter: write the text variable via Default, min 0, max 5000
    Rectangle (946,123 50x30), "Potência"
        OnMouseClick:  Assign=Setup, Type=Assignment
    Rectangle (675,158 22x595)
    Rectangle (841,158 22x595)
    Label (673,158 27x21), "1"
    Label (673,182 27x21), "22"
END_VISUALIZATION

// Dispositivo/Application/Pages/Supervision
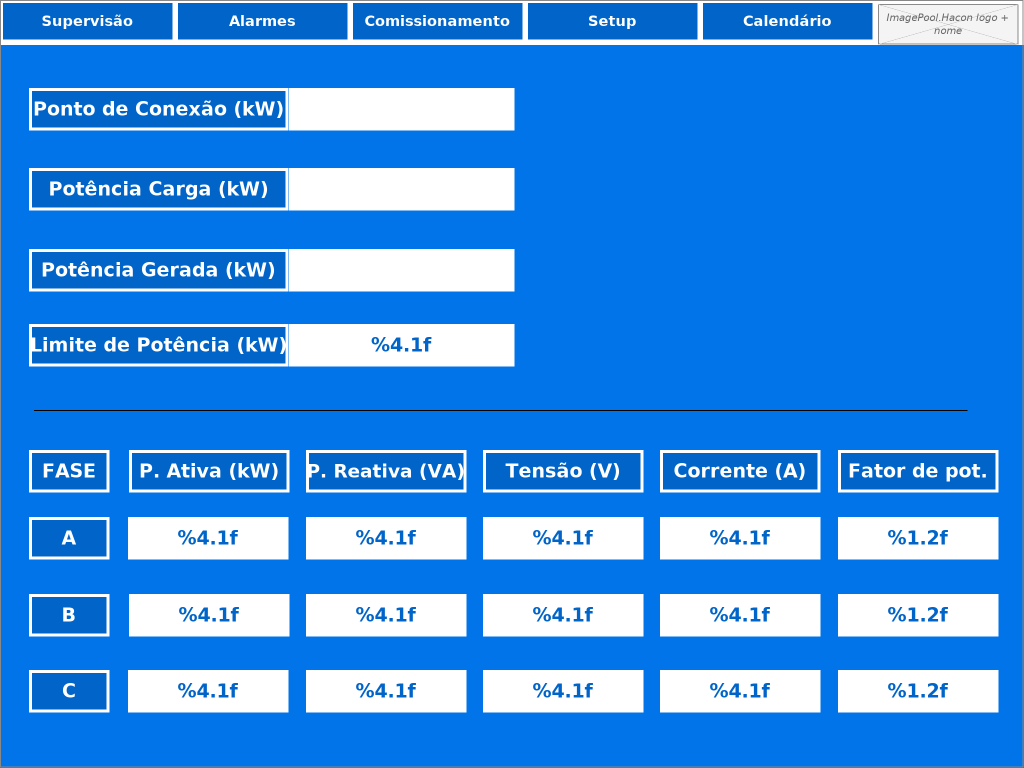
VISUALIZATION Supervision  // 1024x768
    Frame (0,0 1024x768)
        shows Template()
    Rectangle (29,450 80x42), "FASE"
        OnMouseClick:  Assign=Setup, Type=Assignment
    Rectangle (129,450 160x42), "P. Ativa (kW)"
        OnMouseClick:  Assign=Setup, Type=Assignment
    Rectangle (483,450 160x42), "Tensão (V)"
        OnMouseClick:  Assign=Setup, Type=Assignment
    Rectangle (660,450 160x42), "Corrente (A)"
        OnMouseClick:  Assign=Setup, Type=Assignment
    Rectangle (838,450 160x42), "Fator de pot."
        OnMouseClick:  Assign=Setup, Type=Assignment
    Rectangle (29,517 80x42), "A"
        OnMouseClick:  Assign=Setup, Type=Assignment
    Rectangle (29,594 80x42), "B"
        OnMouseClick:  Assign=Setup, Type=Assignment
    Rectangle (29,670 80x42), "C"
        OnMouseClick:  Assign=Setup, Type=Assignment
    Rectangle (128,517 160x42), "%4.1f", text variable: Global.Pa
        OnMouseClick:  Assign=Setup, Type=Assignment
    Line (34,410) (967,410)
    Rectangle (29,88 259x42), "Ponto de Conexão (kW)"
        OnMouseClick:  Assign=Setup, Type=Assignment
    Rectangle (289,88 225x42), "%.1f"
        OnMouseClick:  Assign=Setup, Type=Assignment
    Rectangle (29,168 259x42), "Potência Carga (kW)"
        OnMouseClick:  Assign=Setup, Type=Assignment
    Rectangle (289,168 225x42)
        OnMouseClick:  Assign=Setup, Type=Assignment
    Rectangle (29,249 259x42), "Potência Gerada (kW)"
        OnMouseClick:  Assign=Setup, Type=Assignment
    Rectangle (289,249 225x42)
        OnMouseClick:  Assign=Setup, Type=Assignment
    Rectangle (29,324 259x42), "Limite de Potência (kW)"
        OnMouseClick:  Assign=Setup, Type=Assignment
    Rectangle (289,324 225x42), "%4.1f", text variable: Global.TotalPowerPercent
        OnMouseClick:  Assign=Setup, Type=Assignment
    Rectangle (306,450 160x42), "P. Reativa (VA)"
        OnMouseClick:  Assign=Setup, Type=Assignment
    Rectangle (129,594 160x42), "%4.1f", text variable: Global.Pb
        OnMouseClick:  Assign=Setup, Type=Assignment
    Rectangle (128,670 160x42), "%4.1f", text variable: Global.Pc
        OnMouseClick:  Assign=Setup, Type=Assignment
    Rectangle (306,517 160x42), "%4.1f", text variable: Global.Qa
        OnMouseClick:  Assign=Setup, Type=Assignment
    Rectangle (306,594 160x42), "%4.1f", text variable: Global.Qb
        OnMouseClick:  Assign=Setup, Type=Assignment
    Rectangle (306,670 160x42), "%4.1f", text variable: Global.Qc
        OnMouseClick:  Assign=Setup, Type=Assignment
    Rectangle (483,517 160x42), "%4.1f", text variable: Global.Ua
        OnMouseClick:  Assign=Setup, Type=Assignment
    Rectangle (483,594 160x42), "%4.1f", text variable: Global.Ub
        OnMouseClick:  Assign=Setup, Type=Assignment
    Rectangle (483,670 160x42), "%4.1f", text variable: Global.Uc
        OnMouseClick:  Assign=Setup, Type=Assignment
    Rectangle (660,517 160x42), "%4.1f", text variable: Global.Ia
        OnMouseClick:  Assign=Setup, Type=Assignment
    Rectangle (660,594 160x42), "%4.1f", text variable: Global.Ib
        OnMouseClick:  Assign=Setup, Type=Assignment
    Rectangle (660,670 160x42), "%4.1f", text variable: Global.Ic
        OnMouseClick:  Assign=Setup, Type=Assignment
    Rectangle (838,517 160x42), "%1.2f", text variable: Global.PFa
        OnMouseClick:  Assign=Setup, Type=Assignment
    Rectangle (838,594 160x42), "%1.2f", text variable: Global.PFb
        OnMouseClick:  Assign=Setup, Type=Assignment
    Rectangle (838,670 160x42), "%1.2f", text variable: Global.PFc
        OnMouseClick:  Assign=Setup, Type=Assignment
END_VISUALIZATION

// Dispositivo/Application/Pages/Template
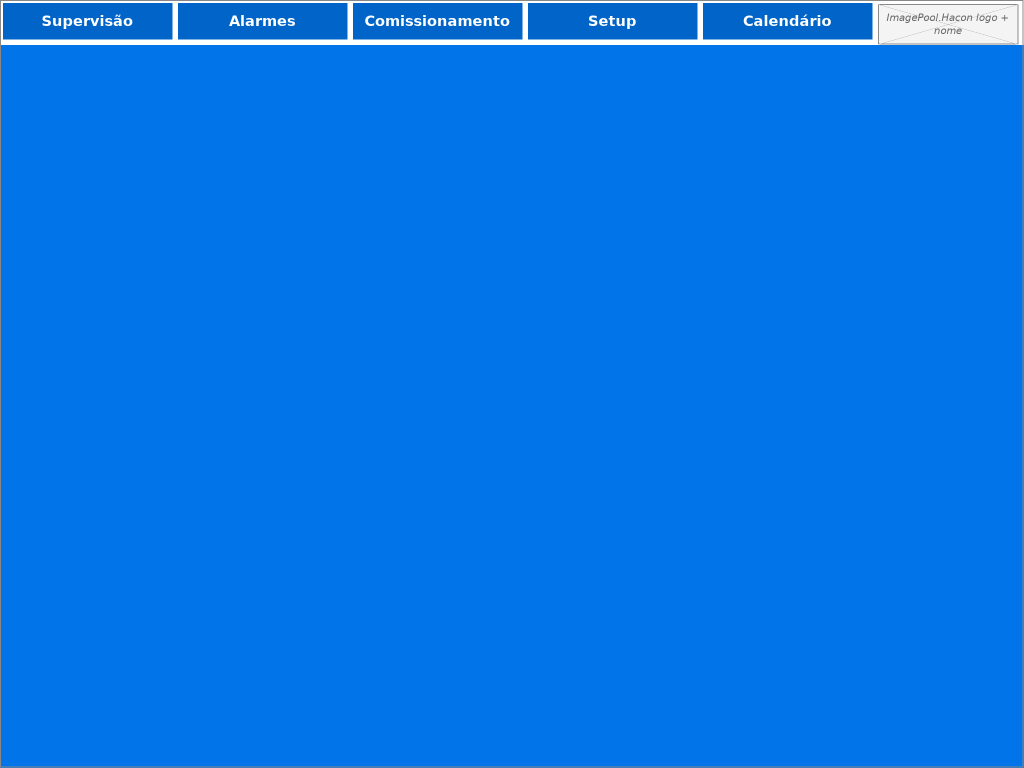
VISUALIZATION Template  // 1024x768
    Rectangle (0,0 1024x768)
    Rectangle (0,0 1024x45)
    Rectangle (0,0 175x42), "Supervisão"
        OnMouseClick:  Assign=Supervision, Type=Assignment
    Rectangle (700,0 175x42), "Calendário"
        OnMouseClick:  Assign=Schedulle, Type=Assignment
    Rectangle (525,0 175x42), "Setup"
        OnMouseClick:  Assign=Setup, Type=Assignment
    Rectangle (350,0 175x42), "Comissionamento"
        OnMouseClick:  Assign=Comissioning, Type=Assignment
    Rectangle (175,0 175x42), "Alarmes"
        OnMouseClick:  Assign=Alarms, Type=Assignment
    Rectangle (0,45 1024x723)
    Image (878,4 140x40), image: ImagePool.Hacon logo + nome
END_VISUALIZATION

// Dispositivo/Application/Pages/Comissioning
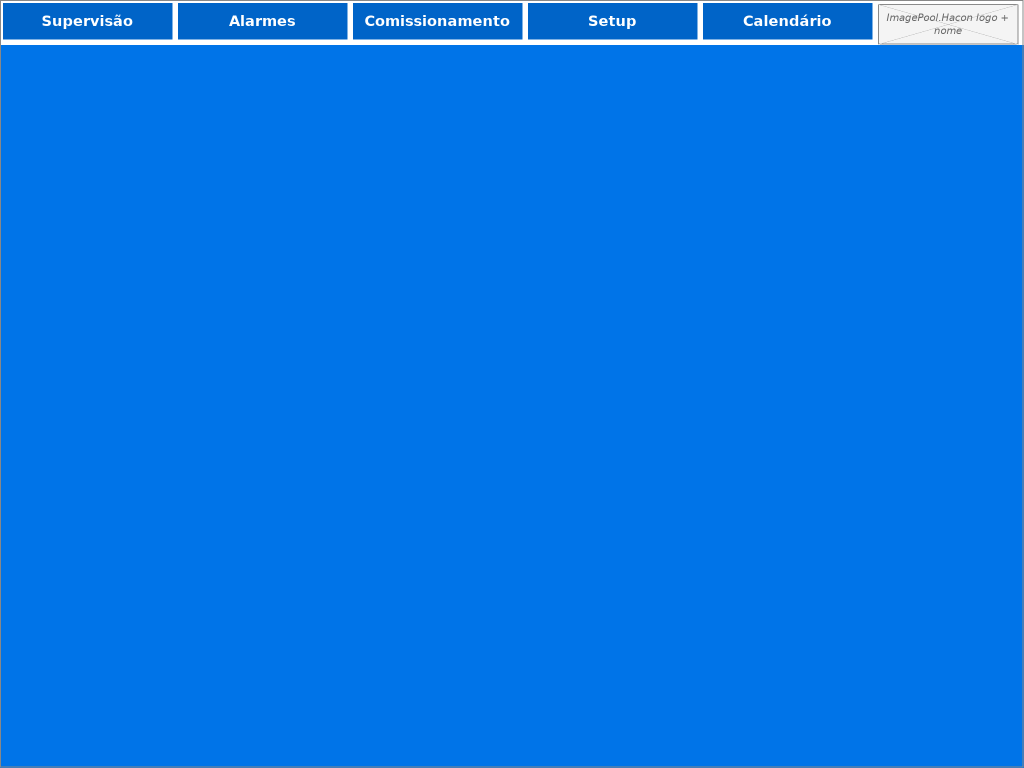
VISUALIZATION Comissioning  // 1024x768
    Frame (0,0 1024x768)
        shows Template()
END_VISUALIZATION

// Dispositivo/Application/Pages/Setup
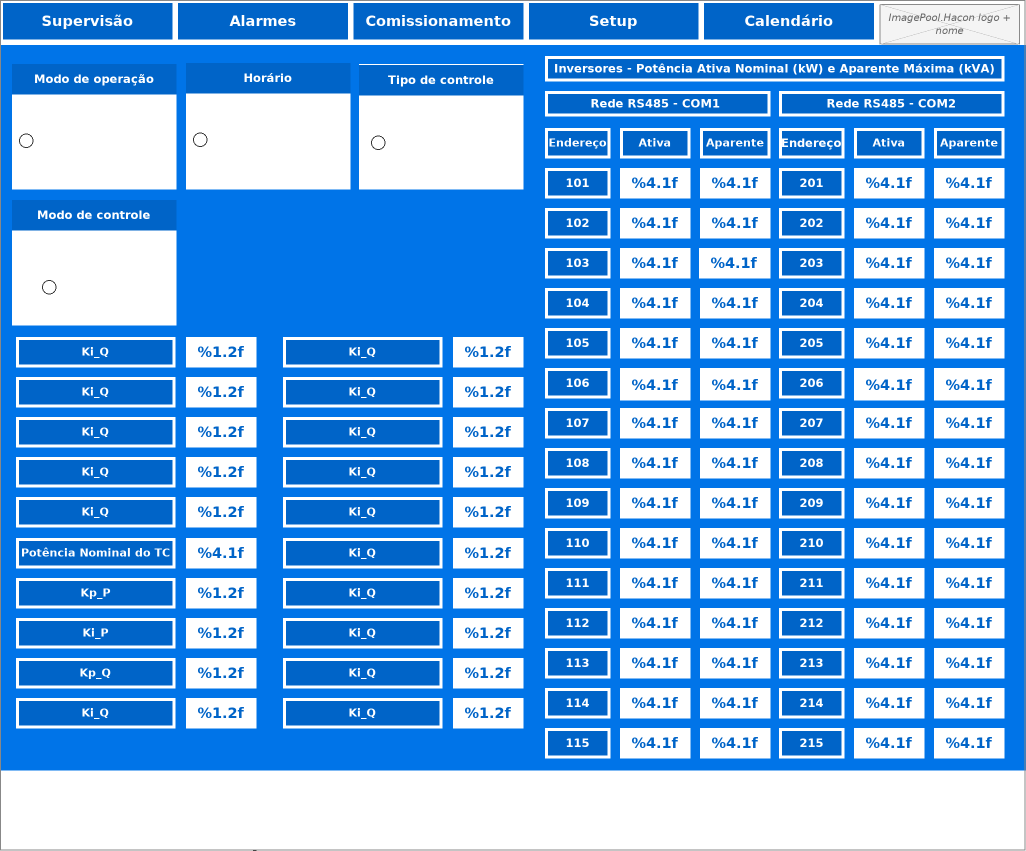
VISUALIZATION Setup  // 1026x851
    Frame (0,0 1026x770)
        shows Template()
    Rectangle (545,168 65x30), "101"
        OnMouseClick:  Assign=Setup, Type=Assignment
    Rectangle (620,168 70x30), "%4.1f", text variable: PerVar.InvActivePower[1]
        OnMouseEnter: write the text variable via Default, min 0, max 5000
    Rectangle (545,128 65x30), "Endereço"
        OnMouseClick:  Assign=Setup, Type=Assignment
    Rectangle (620,128 70x30), "Ativa"
        OnMouseClick:  Assign=Setup, Type=Assignment
    Rectangle (700,128 70x30), "Aparente"
        OnMouseClick:  Assign=Setup, Type=Assignment
    Rectangle (545,56 459x25), "Inversores - Potência Ativa Nominal (kW) e Aparente Máxima (kVA)"
        OnMouseClick:  Assign=Setup, Type=Assignment
    Rectangle (545,208 65x30), "102"
        OnMouseClick:  Assign=Setup, Type=Assignment
    Rectangle (620,208 70x30), text variable: Global.Pa
        OnMouseClick:  Assign=Setup, Type=Assignment
    Rectangle (545,248 65x30), "103"
        OnMouseClick:  Assign=Setup, Type=Assignment
    Rectangle (620,248 70x30), text variable: Global.Pa
        OnMouseClick:  Assign=Setup, Type=Assignment
    Rectangle (545,288 65x30), "104"
        OnMouseClick:  Assign=Setup, Type=Assignment
    Rectangle (620,288 70x30), text variable: Global.Pa
        OnMouseClick:  Assign=Setup, Type=Assignment
    Rectangle (545,328 65x30), "105"
        OnMouseClick:  Assign=Setup, Type=Assignment
    Rectangle (620,328 70x30), text variable: Global.Pa
        OnMouseClick:  Assign=Setup, Type=Assignment
    Rectangle (545,368 65x30), "106"
        OnMouseClick:  Assign=Setup, Type=Assignment
    Rectangle (620,368 70x30), text variable: Global.Pa
        OnMouseClick:  Assign=Setup, Type=Assignment
    Rectangle (545,408 65x30), "107"
        OnMouseClick:  Assign=Setup, Type=Assignment
    Rectangle (620,408 70x30), text variable: Global.Pa
        OnMouseClick:  Assign=Setup, Type=Assignment
    Rectangle (545,448 65x30), "108"
        OnMouseClick:  Assign=Setup, Type=Assignment
    Rectangle (620,448 70x30), text variable: Global.Pa
        OnMouseClick:  Assign=Setup, Type=Assignment
    Rectangle (545,488 65x30), "109"
        OnMouseClick:  Assign=Setup, Type=Assignment
    Rectangle (620,488 70x30), text variable: Global.Pa
        OnMouseClick:  Assign=Setup, Type=Assignment
    Rectangle (545,528 65x30), "110"
        OnMouseClick:  Assign=Setup, Type=Assignment
    Rectangle (620,528 70x30), text variable: Global.Pa
        OnMouseClick:  Assign=Setup, Type=Assignment
    Rectangle (545,568 65x30), "111"
        OnMouseClick:  Assign=Setup, Type=Assignment
    Rectangle (620,568 70x30), text variable: Global.Pa
        OnMouseClick:  Assign=Setup, Type=Assignment
    Rectangle (545,608 65x30), "112"
        OnMouseClick:  Assign=Setup, Type=Assignment
    Rectangle (620,608 70x30), text variable: Global.Pa
        OnMouseClick:  Assign=Setup, Type=Assignment
    Rectangle (545,648 65x30), "113"
        OnMouseClick:  Assign=Setup, Type=Assignment
    Rectangle (620,648 70x30), text variable: Global.Pa
        OnMouseClick:  Assign=Setup, Type=Assignment
    Rectangle (545,688 65x30), "114"
        OnMouseClick:  Assign=Setup, Type=Assignment
    Rectangle (620,688 70x30), text variable: Global.Pa
        OnMouseClick:  Assign=Setup, Type=Assignment
    Rectangle (545,728 65x30), "115"
        OnMouseClick:  Assign=Setup, Type=Assignment
    Rectangle (620,728 70x30), text variable: Global.Pa
        OnMouseClick:  Assign=Setup, Type=Assignment
    Rectangle (545,91 225x25), "Rede RS485 - COM1"
        OnMouseClick:  Assign=Setup, Type=Assignment
    Rectangle (779,91 225x25), "Rede RS485 - COM2"
        OnMouseClick:  Assign=Setup, Type=Assignment
    Rectangle (779,168 65x30), "201"
        OnMouseClick:  Assign=Setup, Type=Assignment
    Rectangle (779,208 65x30), "202"
        OnMouseClick:  Assign=Setup, Type=Assignment
    Rectangle (779,248 65x30), "203"
        OnMouseClick:  Assign=Setup, Type=Assignment
    Rectangle (779,288 65x30), "204"
        OnMouseClick:  Assign=Setup, Type=Assignment
    Rectangle (779,328 65x30), "205"
        OnMouseClick:  Assign=Setup, Type=Assignment
    Rectangle (779,368 65x30), "206"
        OnMouseClick:  Assign=Setup, Type=Assignment
    Rectangle (779,408 65x30), "207"
        OnMouseClick:  Assign=Setup, Type=Assignment
    Rectangle (779,448 65x30), "208"
        OnMouseClick:  Assign=Setup, Type=Assignment
    Rectangle (779,488 65x30), "209"
        OnMouseClick:  Assign=Setup, Type=Assignment
    Rectangle (779,528 65x30), "210"
        OnMouseClick:  Assign=Setup, Type=Assignment
    Rectangle (779,568 65x30), "211"
        OnMouseClick:  Assign=Setup, Type=Assignment
    Rectangle (779,608 65x30), "212"
        OnMouseClick:  Assign=Setup, Type=Assignment
    Rectangle (779,648 65x30), "213"
        OnMouseClick:  Assign=Setup, Type=Assignment
    Rectangle (779,688 65x30), "214"
        OnMouseClick:  Assign=Setup, Type=Assignment
    Rectangle (779,728 65x30), "215"
        OnMouseClick:  Assign=Setup, Type=Assignment
    Rectangle (779,128 65x30), "Endereço"
        OnMouseClick:  Assign=Setup, Type=Assignment
    Rectangle (854,128 70x30), "Ativa"
        OnMouseClick:  Assign=Setup, Type=Assignment
    Rectangle (934,128 70x30), "Aparente"
        OnMouseClick:  Assign=Setup, Type=Assignment
    Rectangle (620,208 70x30), "%4.1f", text variable: PerVar.InvActivePower[2]
        OnMouseEnter: write the text variable via Default, min 0, max 5000
    Rectangle (620,248 70x30), "%4.1f", text variable: PerVar.InvActivePower[3]
        OnMouseEnter: write the text variable via Default, min 0, max 5000
    Rectangle (620,288 70x30), "%4.1f", text variable: PerVar.InvActivePower[4]
        OnMouseEnter: write the text variable via Default, min 0, max 5000
    Rectangle (620,328 70x30), "%4.1f", text variable: PerVar.InvActivePower[5]
        OnMouseEnter: write the text variable via Default, min 0, max 5000
    Rectangle (620,370 70x30), "%4.1f", text variable: PerVar.InvActivePower[6]
        OnMouseEnter: write the text variable via Default, min 0, max 5000
    Rectangle (620,408 70x30), "%4.1f", text variable: PerVar.InvActivePower[7]
        OnMouseEnter: write the text variable via Default, min 0, max 5000
    Rectangle (620,448 70x30), "%4.1f", text variable: PerVar.InvActivePower[8]
        OnMouseEnter: write the text variable via Default, min 0, max 5000
    Rectangle (620,488 70x30), "%4.1f", text variable: PerVar.InvActivePower[9]
        OnMouseEnter: write the text variable via Default, min 0, max 5000
    Rectangle (620,528 70x30), "%4.1f", text variable: PerVar.InvActivePower[10]
        OnMouseEnter: write the text variable via Default, min 0, max 5000
    Rectangle (620,568 70x30), "%4.1f", text variable: PerVar.InvActivePower[11]
        OnMouseEnter: write the text variable via Default, min 0, max 5000
    Rectangle (620,608 70x30), "%4.1f", text variable: PerVar.InvActivePower[12]
        OnMouseEnter: write the text variable via Default, min 0, max 5000
    Rectangle (620,648 70x30), "%4.1f", text variable: PerVar.InvActivePower[13]
        OnMouseEnter: write the text variable via Default, min 0, max 5000
    Rectangle (620,688 70x30), "%4.1f", text variable: PerVar.InvActivePower[14]
        OnMouseEnter: write the text variable via Default, min 0, max 5000
    Rectangle (620,728 70x30), "%4.1f", text variable: PerVar.InvActivePower[15]
        OnMouseEnter: write the text variable via Default, min 0, max 5000
    Rectangle (854,168 70x30), "%4.1f", text variable: PerVar.InvActivePower[16]
        OnMouseEnter: write the text variable via Default, min 0, max 5000
    Rectangle (854,208 70x30), text variable: Global.Pa
        OnMouseClick:  Assign=Setup, Type=Assignment
    Rectangle (854,248 70x30), text variable: Global.Pa
        OnMouseClick:  Assign=Setup, Type=Assignment
    Rectangle (854,288 70x30), text variable: Global.Pa
        OnMouseClick:  Assign=Setup, Type=Assignment
    Rectangle (854,328 70x30), text variable: Global.Pa
        OnMouseClick:  Assign=Setup, Type=Assignment
    Rectangle (854,368 70x30), text variable: Global.Pa
        OnMouseClick:  Assign=Setup, Type=Assignment
    Rectangle (854,408 70x30), text variable: Global.Pa
        OnMouseClick:  Assign=Setup, Type=Assignment
    Rectangle (854,448 70x30), text variable: Global.Pa
        OnMouseClick:  Assign=Setup, Type=Assignment
    Rectangle (854,488 70x30), text variable: Global.Pa
        OnMouseClick:  Assign=Setup, Type=Assignment
    Rectangle (854,528 70x30), text variable: Global.Pa
        OnMouseClick:  Assign=Setup, Type=Assignment
    Rectangle (854,568 70x30), text variable: Global.Pa
        OnMouseClick:  Assign=Setup, Type=Assignment
    Rectangle (854,608 70x30), text variable: Global.Pa
        OnMouseClick:  Assign=Setup, Type=Assignment
    Rectangle (854,648 70x30), text variable: Global.Pa
        OnMouseClick:  Assign=Setup, Type=Assignment
    Rectangle (854,688 70x30), text variable: Global.Pa
        OnMouseClick:  Assign=Setup, Type=Assignment
    Rectangle (854,728 70x30), text variable: Global.Pa
        OnMouseClick:  Assign=Setup, Type=Assignment
    Rectangle (854,208 70x30), "%4.1f", text variable: PerVar.InvActivePower[17]
        OnMouseEnter: write the text variable via Default, min 0, max 5000
    Rectangle (854,248 70x30), "%4.1f", text variable: PerVar.InvActivePower[18]
        OnMouseEnter: write the text variable via Default, min 0, max 5000
    Rectangle (854,288 70x30), "%4.1f", text variable: PerVar.InvActivePower[19]
        OnMouseEnter: write the text variable via Default, min 0, max 5000
    Rectangle (854,328 70x30), "%4.1f", text variable: PerVar.InvActivePower[20]
        OnMouseEnter: write the text variable via Default, min 0, max 5000
    Rectangle (854,370 70x30), "%4.1f", text variable: PerVar.InvActivePower[21]
        OnMouseEnter: write the text variable via Default, min 0, max 5000
    Rectangle (854,408 70x30), "%4.1f", text variable: PerVar.InvActivePower[22]
        OnMouseEnter: write the text variable via Default, min 0, max 5000
    Rectangle (854,448 70x30), "%4.1f", text variable: PerVar.InvActivePower[23]
        OnMouseEnter: write the text variable via Default, min 0, max 5000
    Rectangle (854,488 70x30), "%4.1f", text variable: PerVar.InvActivePower[24]
        OnMouseEnter: write the text variable via Default, min 0, max 5000
    Rectangle (854,528 70x30), "%4.1f", text variable: PerVar.InvActivePower[25]
        OnMouseEnter: write the text variable via Default, min 0, max 5000
    Rectangle (854,568 70x30), "%4.1f", text variable: PerVar.InvActivePower[26]
        OnMouseEnter: write the text variable via Default, min 0, max 5000
    Rectangle (854,608 70x30), "%4.1f", text variable: PerVar.InvActivePower[27]
        OnMouseEnter: write the text variable via Default, min 0, max 5000
    Rectangle (854,648 70x30), "%4.1f", text variable: PerVar.InvActivePower[28]
        OnMouseEnter: write the text variable via Default, min 0, max 5000
    Rectangle (854,688 70x30), "%4.1f", text variable: PerVar.InvActivePower[29]
        OnMouseEnter: write the text variable via Default, min 0, max 5000
    Rectangle (854,728 70x30), "%4.1f", text variable: PerVar.InvActivePower[30]
        OnMouseEnter: write the text variable via Default, min 0, max 5000
    Rectangle (700,208 70x30), text variable: Global.Pa
        OnMouseClick:  Assign=Setup, Type=Assignment
    Rectangle (700,248 70x30), text variable: Global.Pa
        OnMouseClick:  Assign=Setup, Type=Assignment
    Rectangle (700,288 70x30), text variable: Global.Pa
        OnMouseClick:  Assign=Setup, Type=Assignment
    Rectangle (700,328 70x30), text variable: Global.Pa
        OnMouseClick:  Assign=Setup, Type=Assignment
    Rectangle (700,368 70x30), text variable: Global.Pa
        OnMouseClick:  Assign=Setup, Type=Assignment
    Rectangle (700,408 70x30), text variable: Global.Pa
        OnMouseClick:  Assign=Setup, Type=Assignment
    Rectangle (700,448 70x30), text variable: Global.Pa
        OnMouseClick:  Assign=Setup, Type=Assignment
    Rectangle (700,488 70x30), text variable: Global.Pa
        OnMouseClick:  Assign=Setup, Type=Assignment
    Rectangle (700,528 70x30), text variable: Global.Pa
        OnMouseClick:  Assign=Setup, Type=Assignment
    Rectangle (700,568 70x30), text variable: Global.Pa
        OnMouseClick:  Assign=Setup, Type=Assignment
    Rectangle (700,608 70x30), text variable: Global.Pa
        OnMouseClick:  Assign=Setup, Type=Assignment
    Rectangle (700,648 70x30), text variable: Global.Pa
        OnMouseClick:  Assign=Setup, Type=Assignment
    Rectangle (700,688 70x30), text variable: Global.Pa
        OnMouseClick:  Assign=Setup, Type=Assignment
    Rectangle (700,728 70x30), text variable: Global.Pa
        OnMouseClick:  Assign=Setup, Type=Assignment
    Rectangle (700,208 70x30), "%4.1f", text variable: PerVar.InvSmaxPower[2]
        OnMouseEnter: write the text variable via Default, min 0, max 5000
    Rectangle (700,288 70x30), "%4.1f", text variable: PerVar.InvSmaxPower[4]
        OnMouseEnter: write the text variable via Default, min 0, max 5000
    Rectangle (700,328 70x30), "%4.1f", text variable: PerVar.InvSmaxPower[5]
        OnMouseEnter: write the text variable via Default, min 0, max 5000
    Rectangle (700,370 70x30), "%4.1f", text variable: PerVar.InvSmaxPower[6]
        OnMouseEnter: write the text variable via Default, min 0, max 5000
    Rectangle (700,408 70x30), "%4.1f", text variable: PerVar.InvSmaxPower[7]
        OnMouseEnter: write the text variable via Default, min 0, max 5000
    Rectangle (700,448 70x30), "%4.1f", text variable: PerVar.InvSmaxPower[8]
        OnMouseEnter: write the text variable via Default, min 0, max 5000
    Rectangle (700,488 70x30), "%4.1f", text variable: PerVar.InvSmaxPower[9]
        OnMouseEnter: write the text variable via Default, min 0, max 5000
    Rectangle (700,528 70x30), "%4.1f", text variable: PerVar.InvSmaxPower[10]
        OnMouseEnter: write the text variable via Default, min 0, max 5000
    Rectangle (700,568 70x30), "%4.1f", text variable: PerVar.InvSmaxPower[11]
        OnMouseEnter: write the text variable via Default, min 0, max 5000
    Rectangle (700,608 70x30), "%4.1f", text variable: PerVar.InvSmaxPower[12]
        OnMouseEnter: write the text variable via Default, min 0, max 5000
    Rectangle (700,648 70x30), "%4.1f", text variable: PerVar.InvSmaxPower[13]
        OnMouseEnter: write the text variable via Default, min 0, max 5000
    Rectangle (700,688 70x30), "%4.1f", text variable: PerVar.InvSmaxPower[14]
        OnMouseEnter: write the text variable via Default, min 0, max 5000
    Rectangle (700,728 70x30), "%4.1f", text variable: PerVar.InvSmaxPower[15]
        OnMouseEnter: write the text variable via Default, min 0, max 5000
    Rectangle (934,168 70x30), "%4.1f", text variable: PerVar.InvSmaxPower[16]
        OnMouseEnter: write the text variable via Default, min 0, max 5000
    Rectangle (934,208 70x30), text variable: Global.Pa
        OnMouseClick:  Assign=Setup, Type=Assignment
    Rectangle (934,248 70x30), text variable: Global.Pa
        OnMouseClick:  Assign=Setup, Type=Assignment
    Rectangle (934,288 70x30), text variable: Global.Pa
        OnMouseClick:  Assign=Setup, Type=Assignment
    Rectangle (934,328 70x30), text variable: Global.Pa
        OnMouseClick:  Assign=Setup, Type=Assignment
    Rectangle (934,368 70x30), text variable: Global.Pa
        OnMouseClick:  Assign=Setup, Type=Assignment
    Rectangle (934,408 70x30), text variable: Global.Pa
        OnMouseClick:  Assign=Setup, Type=Assignment
    Rectangle (934,448 70x30), text variable: Global.Pa
        OnMouseClick:  Assign=Setup, Type=Assignment
    Rectangle (934,488 70x30), text variable: Global.Pa
        OnMouseClick:  Assign=Setup, Type=Assignment
    Rectangle (934,528 70x30), text variable: Global.Pa
        OnMouseClick:  Assign=Setup, Type=Assignment
    Rectangle (934,568 70x30), text variable: Global.Pa
        OnMouseClick:  Assign=Setup, Type=Assignment
    Rectangle (934,608 70x30), text variable: Global.Pa
        OnMouseClick:  Assign=Setup, Type=Assignment
    Rectangle (934,648 70x30), text variable: Global.Pa
        OnMouseClick:  Assign=Setup, Type=Assignment
    Rectangle (934,688 70x30), text variable: Global.Pa
        OnMouseClick:  Assign=Setup, Type=Assignment
    Rectangle (934,728 70x30), text variable: Global.Pa
        OnMouseClick:  Assign=Setup, Type=Assignment
    Rectangle (934,208 70x30), "%4.1f", text variable: PerVar.InvSmaxPower[17]
        OnMouseEnter: write the text variable via Default, min 0, max 5000
    Rectangle (934,248 70x30), "%4.1f", text variable: PerVar.InvSmaxPower[18]
        OnMouseEnter: write the text variable via Default, min 0, max 5000
    Rectangle (934,288 70x30), "%4.1f", text variable: PerVar.InvSmaxPower[19]
        OnMouseEnter: write the text variable via Default, min 0, max 5000
    Rectangle (934,328 70x30), "%4.1f", text variable: PerVar.InvSmaxPower[20]
        OnMouseEnter: write the text variable via Default, min 0, max 5000
    Rectangle (934,370 70x30), "%4.1f", text variable: PerVar.InvSmaxPower[21]
        OnMouseEnter: write the text variable via Default, min 0, max 5000
    Rectangle (934,408 70x30), "%4.1f", text variable: PerVar.InvSmaxPower[22]
        OnMouseEnter: write the text variable via Default, min 0, max 5000
    Rectangle (934,448 70x30), "%4.1f", text variable: PerVar.InvSmaxPower[23]
        OnMouseEnter: write the text variable via Default, min 0, max 5000
    Rectangle (934,488 70x30), "%4.1f", text variable: PerVar.InvSmaxPower[24]
        OnMouseEnter: write the text variable via Default, min 0, max 5000
    Rectangle (934,528 70x30), "%4.1f", text variable: PerVar.InvSmaxPower[25]
        OnMouseEnter: write the text variable via Default, min 0, max 5000
    Rectangle (934,568 70x30), "%4.1f", text variable: PerVar.InvSmaxPower[26]
        OnMouseEnter: write the text variable via Default, min 0, max 5000
    Rectangle (934,608 70x30), "%4.1f", text variable: PerVar.InvSmaxPower[27]
        OnMouseEnter: write the text variable via Default, min 0, max 5000
    Rectangle (934,648 70x30), "%4.1f", text variable: PerVar.InvSmaxPower[28]
        OnMouseEnter: write the text variable via Default, min 0, max 5000
    Rectangle (934,688 70x30), "%4.1f", text variable: PerVar.InvSmaxPower[29]
        OnMouseEnter: write the text variable via Default, min 0, max 5000
    Rectangle (934,728 70x30), "%4.1f", text variable: PerVar.InvSmaxPower[30]
        OnMouseEnter: write the text variable via Default, min 0, max 5000
    Rectangle (699,248 70x30), "%4.1f", text variable: PerVar.InvSmaxPower[3]
        OnMouseEnter: write the text variable via Default, min 0, max 5000
    Rectangle (700,168 70x30), "%4.1f", text variable: PerVar.InvSmaxPower[1]
        OnMouseEnter: write the text variable via Default, min 0, max 5000
    Rectangle (253,851 3x0)
    Rectangle (12,64 164x125)
    RadioButton (17,105 154x71), variable: PerVar.OperationMode
    Rectangle (186,64 164x125)
    RadioButton (191,104 154x71), variable: PerVar.bHorarioVerao
        Areas[0]: Text=Horário NORMAL
        Areas[1]: Text=Horário de VERÃO
    Rectangle (16,538 159x30), "Potência Nominal do TC"
        OnMouseClick:  Assign=Setup, Type=Assignment
    Rectangle (186,538 70x30), "%4.1f", text variable: PerVar.TC_Power_kW
        OnMouseEnter: write the text variable via Default, min 0, max 5000
    Rectangle (359,64 164x125)
    RadioButton (369,96 154x93), variable: PerVar.PowerMode
        Areas[0]: Text=Total
        Areas[1]: Text=Fase
        Areas[2]: Text=Ambos
    Rectangle (16,578 159x30), "Kp_P"
        OnMouseClick:  Assign=Setup, Type=Assignment
    Rectangle (186,578 70x30), "%1.2f", text variable: PerVar.Kp_P
        OnMouseEnter: write the text variable via Default, min 0, max 5000
    Rectangle (16,618 159x30), "Ki_P"
        OnMouseClick:  Assign=Setup, Type=Assignment
    Rectangle (186,618 70x30), "%1.2f", text variable: PerVar.Ki_P
        OnMouseEnter: write the text variable via Default, min 0, max 5000
    Rectangle (16,658 159x30), "Kp_Q"
        OnMouseClick:  Assign=Setup, Type=Assignment
    Rectangle (186,658 70x30), "%1.2f", text variable: PerVar.Kp_Q
        OnMouseEnter: write the text variable via Default, min 0, max 5000
    Rectangle (16,698 159x30), "Ki_Q"
        OnMouseClick:  Assign=Setup, Type=Assignment
    Rectangle (186,698 70x30), "%1.2f", text variable: PerVar.Ki_Q
        OnMouseEnter: write the text variable via Default, min 0, max 5000
    Rectangle (12,200 164x125)
    RadioButton (40,247 108x80), variable: PerVar.ControlMode
        Areas[0]: Text=Manual
        Areas[1]: Text=Automatico
    Rectangle (12,200 164x30), "Modo de controle"
        OnMouseClick:  Assign=Setup, Type=Assignment
    Rectangle (186,63 164x30), "Horário"
        OnMouseClick:  Assign=Setup, Type=Assignment
    Rectangle (12,64 164x30), "Modo de operação"
        OnMouseClick:  Assign=Setup, Type=Assignment
    Rectangle (359,65 164x30), "Tipo de controle"
        OnMouseClick:  Assign=Setup, Type=Assignment
    Group (283,698 240x30)
        Rectangle (0,0 159x30), "Ki_Q"
            OnMouseClick:  Assign=Setup, Type=Assignment
        Rectangle (170,0 70x30), "%1.2f", text variable: PerVar.Ki_Q
            OnMouseEnter: write the text variable via Default, min 0, max 5000
    Group (283,658 240x30)
        Rectangle (0,0 159x30), "Ki_Q"
            OnMouseClick:  Assign=Setup, Type=Assignment
        Rectangle (170,0 70x30), "%1.2f", text variable: PerVar.Ki_Q
            OnMouseEnter: write the text variable via Default, min 0, max 5000
    Group (283,618 240x30)
        Rectangle (0,0 159x30), "Ki_Q"
            OnMouseClick:  Assign=Setup, Type=Assignment
        Rectangle (170,0 70x30), "%1.2f", text variable: PerVar.Ki_Q
            OnMouseEnter: write the text variable via Default, min 0, max 5000
    Group (283,578 240x30)
        Rectangle (0,0 159x30), "Ki_Q"
            OnMouseClick:  Assign=Setup, Type=Assignment
        Rectangle (170,0 70x30), "%1.2f", text variable: PerVar.Ki_Q
            OnMouseEnter: write the text variable via Default, min 0, max 5000
    Group (283,538 240x30)
        Rectangle (0,0 159x30), "Ki_Q"
            OnMouseClick:  Assign=Setup, Type=Assignment
        Rectangle (170,0 70x30), "%1.2f", text variable: PerVar.Ki_Q
            OnMouseEnter: write the text variable via Default, min 0, max 5000
    Group (16,497 240x30)
        Rectangle (0,0 159x30), "Ki_Q"
            OnMouseClick:  Assign=Setup, Type=Assignment
        Rectangle (170,0 70x30), "%1.2f", text variable: PerVar.Ki_Q
            OnMouseEnter: write the text variable via Default, min 0, max 5000
    Group (16,457 240x30)
        Rectangle (0,0 159x30), "Ki_Q"
            OnMouseClick:  Assign=Setup, Type=Assignment
        Rectangle (170,0 70x30), "%1.2f", text variable: PerVar.Ki_Q
            OnMouseEnter: write the text variable via Default, min 0, max 5000
    Group (16,417 240x30)
        Rectangle (0,0 159x30), "Ki_Q"
            OnMouseClick:  Assign=Setup, Type=Assignment
        Rectangle (170,0 70x30), "%1.2f", text variable: PerVar.Ki_Q
            OnMouseEnter: write the text variable via Default, min 0, max 5000
    Group (16,377 240x30)
        Rectangle (0,0 159x30), "Ki_Q"
            OnMouseClick:  Assign=Setup, Type=Assignment
        Rectangle (170,0 70x30), "%1.2f", text variable: PerVar.Ki_Q
            OnMouseEnter: write the text variable via Default, min 0, max 5000
    Group (16,337 240x30)
        Rectangle (0,0 159x30), "Ki_Q"
            OnMouseClick:  Assign=Setup, Type=Assignment
        Rectangle (170,0 70x30), "%1.2f", text variable: PerVar.Ki_Q
            OnMouseEnter: write the text variable via Default, min 0, max 5000
    Group (283,497 240x30)
        Rectangle (0,0 159x30), "Ki_Q"
            OnMouseClick:  Assign=Setup, Type=Assignment
        Rectangle (170,0 70x30), "%1.2f", text variable: PerVar.Ki_Q
            OnMouseEnter: write the text variable via Default, min 0, max 5000
    Group (283,457 240x30)
        Rectangle (0,0 159x30), "Ki_Q"
            OnMouseClick:  Assign=Setup, Type=Assignment
        Rectangle (170,0 70x30), "%1.2f", text variable: PerVar.Ki_Q
            OnMouseEnter: write the text variable via Default, min 0, max 5000
    Group (283,417 240x30)
        Rectangle (0,0 159x30), "Ki_Q"
            OnMouseClick:  Assign=Setup, Type=Assignment
        Rectangle (170,0 70x30), "%1.2f", text variable: PerVar.Ki_Q
            OnMouseEnter: write the text variable via Default, min 0, max 5000
    Group (283,377 240x30)
        Rectangle (0,0 159x30), "Ki_Q"
            OnMouseClick:  Assign=Setup, Type=Assignment
        Rectangle (170,0 70x30), "%1.2f", text variable: PerVar.Ki_Q
            OnMouseEnter: write the text variable via Default, min 0, max 5000
    Group (283,337 240x30)
        Rectangle (0,0 159x30), "Ki_Q"
            OnMouseClick:  Assign=Setup, Type=Assignment
        Rectangle (170,0 70x30), "%1.2f", text variable: PerVar.Ki_Q
            OnMouseEnter: write the text variable via Default, min 0, max 5000
END_VISUALIZATION

(* text list System (id | default)
  Apr | Apr
  April | April
  Aug | Aug
  August | August
  Dec | Dec
  December | December
  Feb | Feb
  February | February
  Fri | Fri
  Friday | Friday
  Jan | Jan
  January | January
  Jul | Jul
  July | July
  Jun | Jun
  June | June
  Mar | Mar
  March | March
  May | May
  May_3Letter | May
  Mon | Mon
  Monday | Monday
  Nov | Nov
  November | November
  Oct | Oct
  October | October
  Sat | Sat
  Saturday | Saturday
  Sep | Sep
  September | September
  Sun | Sun
  Sunday | Sunday
  Thu | Thu
  Thursday | Thursday
  Tue | Tue
  Tuesday | Tuesday
  Wed | Wed
  Wednesday | Wednesday
   |  *)

(* text list Startup (id | default)
  0 | 
   |  *)

(* text list Measurement (id | default)
   |  *)

(* text list InverterComms (id | default)
   |  *)

(* text list Protection (id | default)
   |  *)

(* text list StopTrip (id | default)
   |  *)

(* text list SystemWatchdog (id | default)
   |  *)
